FUNCTION_BLOCK EL5032
VAR
	_io : EL5032_Data;
	{attribute addProperty Name "WcState"}
	_wcState : WcStateInputToggle;
	{attribute addProperty Name "Info data"}
	_infoData : InfoDataAdsDC;
END_VAR

PROPERTY IO : REFERENCE TO EL5032_Data
GET
IO REF= _io;
END_GET
END_PROPERTY

PROPERTY WcState : REFERENCE TO WcStateInputToggle
GET
WcState REF= _wcState;
END_GET
END_PROPERTY

END_FUNCTION_BLOCK

(* stored: Version 1.1.0.1, ProductVersion 3.1.4024.9
   POU EL5032: Id {5df5ba9f-87c0-04cf-24eb-af68c8e96dbb}, SpecialFunc None
   Property IO: Id {461b1b9f-dab3-053d-391b-48d39b291e56}
   Get Get: Id {4a31f5d1-ad95-0000-0ecb-5076435ff80d}
   Property WcState: Id {a3e61491-658b-0072-2f55-149918791a45}
   Get Get: Id {b8be0cf3-8e1a-02cc-333e-d0513c6cf941} *)
